ABB RAPID module: 00624BE6

MODULE ExternalGuidedMotion
    CONST egm_minmax egm_minmax_lin1:=[-1,1]; !in mm
    CONST egm_minmax egm_minmax_rot1:=[-2,2];! in degees

    VAR robtarget startPoint:=[[451, -481, 700],[0.23679, -0.06616, 0.96930, -0.00468],[-1,-2,0,1],[9E9,9E9,9E9,9E9,9E9,9E9]];
    VAR pose posecorTopOfRamp:=[[451, -481, 700],[0.23679, -0.06616, 0.96930, -0.00468]];
    VAR pose object;
    VAR egmident egmID1;
    VAR egmstate egmSt1;

    TASK PERS tooldata tSuctionCup:=[TRUE,[[120,0,57],[0.707106624,-0.000000155,-0.000000251,0.707106939]],[1,[0,0,1],[1,0,0,0],0,0,0]];
    TASK PERS wobjdata TopOfRamp:=[FALSE,TRUE,"",[[0,0,0],[1,0,0,0]],[[451, -481, 700],[0.258819, 0, 0.965926, 0]]];

    PROC main()
        object.rot:= OrientZYX(0, 150, 0); !In relation to the base of the robot. Y is rotated 90 degrees + angle
        TopOfRamp:= [FALSE,TRUE,"",[[0,0,0],[1,0,0,0]],[[451, -481, 700], object.rot]];
        posecorTopOfRamp.rot:= object.rot;
        startPoint.rot:= object.rot;

        MoveJ startPoint,v100,fine,tSuctionCup;
        SetUpEGM;
    ENDPROC


    PROC SetUpEGM()
        EGMReset egmID1;
        EGMGetId egmID1;
        egmSt1 := EGMGetState(egmID1);
        TPWrite "EGM state: "\Num := egmSt1;

        IF egmSt1 <= EGM_STATE_CONNECTED THEN
            ! Set up the EGM data source: UdpUc server using device "EGMsensor:"and configuration "default"
            EGMSetupUC ROB_1, egmID1, "default", "EGMSensor:" \pose;
        ENDIF

        runEGM;

        IF egmSt1 = EGM_STATE_CONNECTED THEN
            TPWrite "Reset EGM instance egmID1";
            EGMReset egmID1;
        ENDIF
    ENDPROC


    PROC runEGM()
        EGMActPose egmID1\Tool:=tSuctionCup \WObj:=TopOfRamp,posecorTopOfRamp ,EGM_FRAME_WORLD, posecorTopOfRamp, EGM_FRAME_WORLD
        \x:=egm_minmax_lin1 \y:=egm_minmax_lin1 \z:=egm_minmax_lin1
        \rx:=egm_minmax_rot1 \ry:=egm_minmax_rot1 \rz:=egm_minmax_rot1\LpFilter:=2\Samplerate:=4\MaxSpeedDeviation:= 5000;

        EGMRunPose egmID1, EGM_STOP_HOLD\x \y \z\CondTime:=20 \RampInTime:=0.5\RampOutTime:=0.5;
        egmSt1:=EGMGetState(egmID1);
    ENDPROC

ENDMODULE
